// TIA Portal V16 export
// export: Created 2024-09-05T15:58:42.7042153Z, ExportSetting WithDefaults, DisplayName Totally Integrated Automation Portal, DisplayVersion V16 Update 6, DisplayName TIA Portal Version Control Interface, DisplayVersion V16 Update 2, DisplayName TIA Portal Openness, DisplayVersion V16 Update 6, DisplayName STEP 7 Professional, DisplayVersion V16 Update 6, DisplayName STEP 7 Safety, DisplayVersion V16, DisplayName WinCC Advanced, DisplayVersion V16 Update 6
VAR_GLOBAL   // PLC tag table "DM_RT"
   "DM_RT-TriggerEnable" AT %Q7.0 : Bool;
   "DM_RT-Trigger" AT %Q7.1 : Bool;
   "DM_RT-TriggerReady" AT %I14.0 : Bool;
   "DM_RT-TriggerAck" AT %I14.1 : Bool;
   "DM_RT-Acquiring" AT %I14.2 : Bool;
   "DM_RT-MissedAcq" AT %I14.3 : Bool;
   "DM_RT-TriggerID" AT %IW15 : Word;
   "DM_RT-BufferResultsEnable" AT %Q8.0 : Bool;
   "DM_RT-ResultsAck" AT %Q8.1 : Bool;
   "DM_RT-Decoding" AT %I9.0 : Bool;
   "DM_RT-Decode Complete" AT %I9.1 : Bool;
   "DM_RT-Results Buffer Overrun" AT %I9.2 : Bool;
   "DM_RT-Results Available" AT %I9.3 : Bool;
   "DM_RT-General Fault" AT %I9.7 : Bool;
   "DM_RT-Train Code" AT %Q9.0 : Bool;
   "DM_RT-Train Match String" AT %Q9.1 : Bool;
   "DM_RT-Train Focus" AT %Q9.2 : Bool;
   "DM_RT-Train Brightness" AT %Q9.3 : Bool;
   "DM_RT-Untrain" AT %Q9.4 : Bool;
   "DM_RT-Execute DMCC" AT %Q9.6 : Bool;
   "DM_RT-Set Match String" AT %Q9.7 : Bool;
   "DM_RT-Train Code Ack" AT %I17.0 : Bool;
   "DM_RT-Train Match String Ack" AT %I17.1 : Bool;
   "DM_RT-Train Focus Ack" AT %I17.2 : Bool;
   "DM_RT-Train Brightness Ack" AT %I17.3 : Bool;
   "DM_RT-Untrain Ack" AT %I17.4 : Bool;
   "DM_RT-Execute DMCC Ack" AT %I17.6 : Bool;
   "DM_RT-Set Match String Ack" AT %I17.7 : Bool;
   "DM_RT-UserData Option" AT %QW208 : Word;
   "DM_RT-UserData Length" AT %QW210 : Word;
   "DM_RT-UserData[0]" AT %QB212 : Byte;
   "DM_RT-UserData[1]" AT %QB213 : Byte;
   "DM_RT-UserData[2]" AT %QB214 : Byte;
   "DM_RT-UserData[3]" AT %QB215 : Byte;
   "DM_RT-UserData[4]" AT %QB216 : Byte;
   "DM_RT-UserData[5]" AT %QB217 : Byte;
   "DM_RT-UserData[6]" AT %QB218 : Byte;
   "DM_RT-UserData[7]" AT %QB219 : Byte;
   "DM_RT-UserData[8]" AT %QB220 : Byte;
   "DM_RT-UserData[9]" AT %QB221 : Byte;
   "DM_RT-UserData[10]" AT %QB222 : Byte;
   "DM_RT-UserData[11]" AT %QB223 : Byte;
   "DM_RT-UserData[12]" AT %QB224 : Byte;
   "DM_RT-UserData[13]" AT %QB225 : Byte;
   "DM_RT-UserData[14]" AT %QB226 : Byte;
   "DM_RT-UserData[15]" AT %QB227 : Byte;
   "DM_RT-ResultID" AT %IW208 : Word;
   "DM_RT-Result Code" AT %IW210 : Word;
   "DM_RT-Result Extended" AT %IW212 : Word;
   "DM_RT-Result Length" AT %IW214 : Word;
   "DM_RT-InspectionResults[0]" AT %IB216 : Byte;
   "DM_RT-InspectionResults[1]" AT %IB217 : Byte;
   "DM_RT-InspectionResults[2]" AT %IB218 : Byte;
   "DM_RT-InspectionResults[3]" AT %IB219 : Byte;
   "DM_RT-InspectionResults[4]" AT %IB220 : Byte;
   "DM_RT-InspectionResults[5]" AT %IB221 : Byte;
   "DM_RT-InspectionResults[6]" AT %IB222 : Byte;
   "DM_RT-InspectionResults[7]" AT %IB223 : Byte;
   "DM_RT-InspectionResults[8]" AT %IB224 : Byte;
   "DM_RT-InspectionResults[9]" AT %IB225 : Byte;
   "DM_RT-InspectionResults[10]" AT %IB226 : Byte;
   "DM_RT-InspectionResults[11]" AT %IB227 : Byte;
   "DM_RT-InspectionResults[12]" AT %IB228 : Byte;
   "DM_RT-InspectionResults[13]" AT %IB229 : Byte;
   "DM_RT-InspectionResults[14]" AT %IB230 : Byte;
   "DM_RT-InspectionResults[15]" AT %IB231 : Byte;
END_VAR
